Staubli VAL3: uniVALClean.pjx

Parameters version=s7.4 stackSize=5000 millimeterUnit=true
Program file=start.pgx
Program file=stop.pgx
Data file=uniVALClean.dtx
Library alias=lib path=./uniVALProtect.zip password=d5a8e388f0bba1da1d5aae9b562b5403
